// TIA Portal V19 export
TYPE "MES_Msg_Send_Err"
   STRUCT
      TimeOut_ACK { ExternalAccessible := 'False'; ExternalVisible := 'False'; ExternalWritable := 'False'} : Bool;
      Buffer_Pop : Struct
         Presence : Bool;
         Code : DInt;
      END_STRUCT;
      Msg_NotAccepted : "MES_Err_&_Msg";
   END_STRUCT;
END_TYPE
